FUNCTION FN_IntraloxToLane : cLaneSel
VAR_INPUT
	IntraloxLane: DINT;
	LaneConfig: Cmp3LaneSwitchMainConfig;
END_VAR

IF LaneConfig.OutGreenLine = IntraloxLane THEN
	FN_IntraloxToLane := cLaneSel.Green;
ELSIF LaneConfig.OutRedLine = IntraloxLane THEN
	FN_IntraloxToLane := cLaneSel.Red;
ELSIF LaneConfig.OutBlueLine = IntraloxLane THEN
	FN_IntraloxToLane := cLaneSel.Blue;
END_IF

END_FUNCTION

(* stored: Version 1.1.0.1, ProductVersion 3.1.4024.6
   POU FN_IntraloxToLane: Id {feea6535-641a-40ac-9464-13e8e864558c}, SpecialFunc None *)
